Omron CX-Programmer project NewProject (CX-Programmer 9.50)

# PLC NewPLC1: CJ1M CPU11
I/O table (CPU CJ1M-CPU11): rack 0 slot 0 CJ1W-ETN21(ETN21Mode); rack 0 slot 1 CJ1W-ID211; rack 0 slot 2 CJ1W-ID211; rack 0 slot 3 CJ1W-OC211; rack 0 slot 4 CJ1W-MAD42

## Global symbols (name address type ; comment)
0.00 BOOL  ; ON
0.01 BOOL  ; OFF
2000.00 BOOL  ; Enable Output 1
2000.04 BOOL  ; Enable Input 1
W0.01 BOOL  ; ON

## Program NewProgram1 (cyclic task 0)
Local symbols
p_on BOOL

### Section Section1

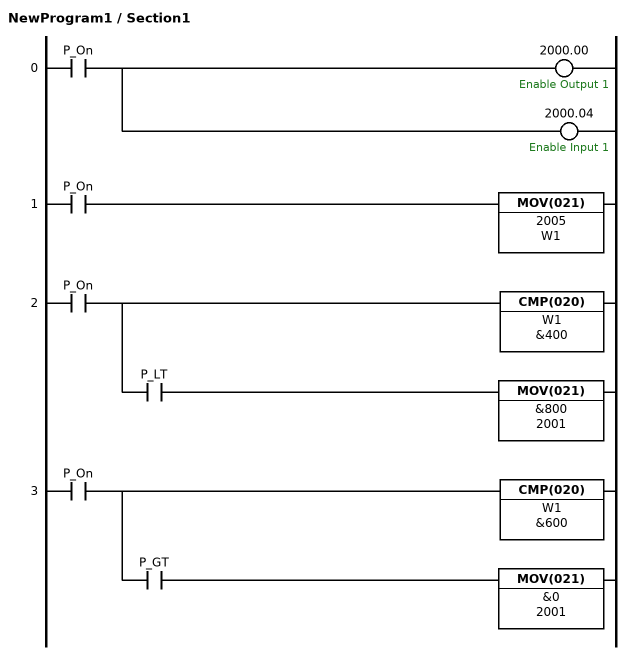
; rung 0
LD P_On
OUT 2000.00  ; Enable Output 1
OUT 2000.04  ; Enable Input 1
; rung 1
LD P_On
MOV(021) 2005 W1
; rung 2
LD P_On
CMP(020) W1 &400
AND P_LT
MOV(021) &800 2001
; rung 3
LD P_On
CMP(020) W1 &600
AND P_GT
MOV(021) &0 2001

### Section END
; rung 0
END(001)